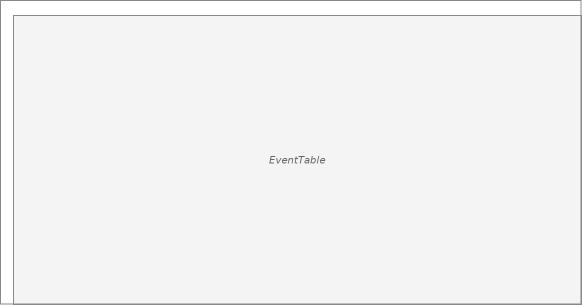
VISUALIZATION Visualization  // 582x305
    EventTable (13,15 569x290)
        p1690906150: Class
        p3258520714: Date
        p2231227367: Time
        p3993844394: Message
        p2076579579: Details
        p3558512729: GVL_EventsSimple.aEventsSimple
        p3921149237: m_pDataArray..pArray
END_VISUALIZATION

(* stored: Version 1.1.0.1, ProductVersion 3.1.4024.3
   Visu Visualization: Id {7bee937a-24ef-4269-b41c-ea5413ee0adc} *)
